// TIA Portal V18 export
VAR_GLOBAL   // PLC tag table "Alarm"
   Trip_TF_Pump_Aeration_Clarifier_01 AT %I0.3 : Bool;
   Trip_TF_Pump_Aeration_Clarifier_02 AT %I0.4 : Bool;
   Trip_Suction_Pump_01 AT %I0.5 : Bool;
   Trip_Suction_Pump_02 AT %I0.6 : Bool;
   Trip_Suction_Pump_03 AT %I0.7 : Bool;
   Trip_Suction_Pump_04 AT %I1.0 : Bool;
   Trip_Suction_Pump_05 AT %I1.1 : Bool;
   Trip_Suction_Pump_06 AT %I1.2 : Bool;
   Trip_Suction_Pump_07 AT %I1.3 : Bool;
   Trip_Suction_Pump_08 AT %I1.4 : Bool;
   Trip_Backwash_Pump_01 AT %I1.5 : Bool;
   Trip_Backwash_Pump_02 AT %I1.6 : Bool;
   Trip_Backwash_Pump_03 AT %I1.7 : Bool;
   Trip_Backwash_Pump_04 AT %I2.0 : Bool;
   Trip_Backwash_Pump_05 AT %I2.1 : Bool;
   Trip_MBR_Aeration_01 AT %I2.2 : Bool;
   Trip_MBR_Aeration_02 AT %I2.3 : Bool;
   Trip_Chlorine_Dosing_Pump AT %I2.4 : Bool;
   Trip_Chlorine_Chemical_Agitator AT %I2.5 : Bool;
   Trip_Solid_TF_Clarifier AT %I2.6 : Bool;
   Trip_UV_1P_01 AT %I2.7 : Bool;
   Trip_UV_1P_02 AT %I3.0 : Bool;
   Trip_UV_1P_03 AT %I3.1 : Bool;
   Trip_TF_Pump_CSAS_B_01 AT %I3.2 : Bool;
   Trip_TF_Pump_CSAS_B_02 AT %I3.3 : Bool;
   Trip_TF_Pump_Aeration_01 AT %I3.4 : Bool;
   Trip_TF_Pump_Aeration_02 AT %I3.5 : Bool;
   Trip_TF_Pump_RWT_MMF_01 AT %I3.6 : Bool;
   Trip_TF_Pump_RWT_MMF_02 AT %I3.7 : Bool;
   Trip_TF_Pump_Waterpool_Buffer_01 AT %I4.0 : Bool;
   Trip_TF_Pump_Waterpool_Buffer_02 AT %I4.1 : Bool;
   Trip_PAC_Flocculant_Dosing_Pump AT %I4.2 : Bool;
   Buzzer AT %Q0.3 : Bool;
END_VAR
